  MoveL 10727 to (516.24, 531.44, 196) mm, rotated rx 180 ry 0 rz 160 deg; joints [9.799, 52.22, -5.839, -141.654, 53.227, 154.66]
  Set speed (17.9 mm/s)
  Call Extruder(1433.21511)
  MoveL 10728 to (515.75, 531.68, 196) mm, rotated rx -180 ry 0 rz 160 deg; joints [9.838, 52.138, -5.688, -141.642, 53.298, 154.686]
  Set speed (17.9 mm/s)
  Call Extruder(1436.45170)
  MoveL 10729 to (514.83, 532.12, 196) mm, rotated rx 180 ry 0 rz 160 deg; joints [9.91, 51.981, -5.403, -141.62, 53.429, 154.738]
  Set speed (17.9 mm/s)
  Call Extruder(1440.77463)
  MoveL 10730 to (513.57, 532.68, 196) mm, rotated rx -180 ry 0 rz 160 deg; joints [10.002, 51.769, -5.017, -141.596, 53.605, 154.81]
  Set speed (17.9 mm/s)
  Call Extruder(1445.24376)
  MoveL 10731 to (512.25, 533.19, 196) mm, rotated rx -180 ry 0 rz 160 deg; joints [10.092, 51.546, -4.609, -141.579, 53.788, 154.892]
  Set speed (17.9 mm/s)
  Call Extruder(1449.94818)
  MoveL 10732 to (510.84, 533.68, 196) mm, rotated rx 180 ry 0 rz 160 deg; joints [10.181, 51.306, -4.172, -141.568, 53.98, 154.985]
  Set speed (17.9 mm/s)
  Call Extruder(1452.28530)
  MoveL 10733 to (510.14, 533.89, 196) mm, rotated rx 180 ry 0 rz 160 deg; joints [10.223, 51.185, -3.952, -141.567, 54.075, 155.034]
  Set speed (17.9 mm/s)
  Call Extruder(1454.80660)
  MoveL 10734 to (509.37, 534.12, 196) mm, rotated rx 180 ry 0 rz 160 deg; joints [10.266, 51.054, -3.714, -141.566, 54.177, 155.088]
  Set speed (17.9 mm/s)
  Call Extruder(1459.03894)
  MoveL 10735 to (508.07, 534.45, 196) mm, rotated rx 180 ry 0 rz 160 deg; joints [10.335, 50.831, -3.309, -141.571, 54.349, 155.182]
  Set speed (17.9 mm/s)
  Call Extruder(1463.69218)
  MoveL 10736 to (506.63, 534.75, 196) mm, rotated rx -180 ry 0 rz 160 deg; joints [10.404, 50.584, -2.858, -141.584, 54.537, 155.292]
  Call Extruder(1468.33973)
  MoveL 10737 to (505.18, 535, 196) mm, rotated rx -180 ry 0 rz 160 deg; joints [10.467, 50.333, -2.403, -141.605, 54.724, 155.408]
  Call Extruder(1472.73701)
  MoveL 10738 to (503.8, 535.18, 196) mm, rotated rx -180 ry 0 rz 160 deg; joints [10.52, 50.094, -1.969, -141.631, 54.898, 155.523]
  Set speed (17.9 mm/s)
  Call Extruder(1477.45397)
  MoveL 10739 to (502.31, 535.3, 196) mm, rotated rx 180 ry 0 rz 160 deg; joints [10.569, 49.836, -1.5, -141.668, 55.084, 155.651]
  Set speed (17.9 mm/s)
  Call Extruder(1482.07202)
  MoveL 10740 to (500.85, 535.37, 196) mm, rotated rx 180 ry 0 rz 160 deg; joints [10.611, 49.582, -1.039, -141.711, 55.264, 155.781]
  Set speed (17.9 mm/s)
  Call Extruder(1486.54739)
  MoveL 10741 to (499.43, 535.38, 196) mm, rotated rx 180 ry 0 rz 160 deg; joints [10.644, 49.334, -0.59, -141.76, 55.436, 155.911]
  Set speed (10.0 mm/s)
  MoveL 10742 to (499.43, 535.38, 200) mm, rotated rx -180 ry 0 rz 160 deg; joints [10.644, 48.828, -0.582, -141.545, 55.045, 155.535]
  Set speed (120.0 mm/s)
  MoveL 10743 to (500.03, 535.97, 200) mm, rotated rx 180 ry 0 rz 160 deg; joints [10.704, 48.952, -0.806, -141.436, 54.992, 155.421]
  Set speed (19.5 mm/s)
  Call Extruder(1491.54324)
  MoveL 10744 to (498.3, 535.93, 200) mm, rotated rx 180 ry 0 rz 160 deg; joints [10.739, 48.648, -0.258, -141.503, 55.197, 155.584]
  Set speed (19.5 mm/s)
  Call Extruder(1494.78231)
  MoveL 10745 to (497.19, 535.86, 200) mm, rotated rx 180 ry 0 rz 160 deg; joints [10.756, 48.451, 0.097, -141.552, 55.328, 155.693]
  Set speed (19.5 mm/s)
  Call Extruder(1496.49093)
  MoveL 10746 to (496.6, 535.81, 200) mm, rotated rx -180 ry 0 rz 160 deg; joints [10.764, 48.347, 0.284, -141.579, 55.396, 155.751]
  Call Extruder(1498.85251)
  MoveL 10747 to (495.79, 535.72, 200) mm, rotated rx -180 ry 0 rz 160 deg; joints [10.772, 48.203, 0.543, -141.619, 55.489, 155.832]
  Set speed (19.5 mm/s)
  Call Extruder(1502.36924)
  MoveL 10748 to (494.59, 535.56, 200) mm, rotated rx -180 ry 0 rz 160 deg; joints [10.781, 47.99, 0.927, -141.682, 55.627, 155.955]
  Set speed (19.5 mm/s)
  Call Extruder(1507.13102)
  MoveL 10749 to (492.97, 535.28, 200) mm, rotated rx 180 ry 0 rz 160 deg; joints [10.784, 47.702, 1.445, -141.776, 55.809, 156.126]
  Set speed (19.5 mm/s)
  Call Extruder(1511.94509)
  MoveL 10750 to (491.35, 534.91, 200) mm, rotated rx -180 ry 0 rz 160 deg; joints [10.777, 47.412, 1.966, -141.88, 55.987, 156.302]
  Set speed (19.5 mm/s)
  Call Extruder(1515.30668)
  MoveL 10751 to (490.22, 534.61, 200) mm, rotated rx 180 ry 0 rz 160 deg; joints [10.766, 47.21, 2.328, -141.958, 56.109, 156.428]
  Set speed (19.5 mm/s)
  Call Extruder(1516.82836)
  MoveL 10752 to (489.72, 534.47, 200) mm, rotated rx 180 ry 0 rz 160 deg; joints [10.76, 47.12, 2.491, -141.995, 56.164, 156.485]
  Call Extruder(1519.31802)
  MoveL 10753 to (488.9, 534.21, 200) mm, rotated rx -180 ry 0 rz 160 deg; joints [10.747, 46.972, 2.756, -142.058, 56.251, 156.58]
  Set speed (19.5 mm/s)
  Call Extruder(1522.70288)
  MoveL 10754 to (487.79, 533.84, 200) mm, rotated rx -180 ry 0 rz 160 deg; joints [10.726, 46.772, 3.114, -142.145, 56.368, 156.71]
  Set speed (19.5 mm/s)
  Call Extruder(1527.20077)
  MoveL 10755 to (486.34, 533.28, 200) mm, rotated rx -180 ry 0 rz 160 deg; joints [10.69, 46.509, 3.586, -142.27, 56.518, 156.885]
  Set speed (19.5 mm/s)
  Call Extruder(1532.16103)
  MoveL 10756 to (484.77, 532.59, 200) mm, rotated rx 180 ry 0 rz 160 deg; joints [10.64, 46.223, 4.098, -142.417, 56.678, 157.081]
  Set speed (19.5 mm/s)
  Call Extruder(1535.74782)
  MoveL 10757 to (483.66, 532.04, 200) mm, rotated rx -180 ry 0 rz 160 deg; joints [10.597, 46.019, 4.463, -142.528, 56.789, 157.225]
  Set speed (19.5 mm/s)
  Call Extruder(1537.52530)
  MoveL 10758 to (483.11, 531.76, 200) mm, rotated rx 180 ry 0 rz 160 deg; joints [10.574, 45.919, 4.642, -142.585, 56.843, 157.296]
  Set speed (19.5 mm/s)
  Call Extruder(1539.75504)
  MoveL 10759 to (482.44, 531.39, 200) mm, rotated rx -180 ry 0 rz 160 deg; joints [10.542, 45.794, 4.865, -142.659, 56.908, 157.386]
  Set speed (19.5 mm/s)
  Call Extruder(1543.11777)
  MoveL 10760 to (481.43, 530.81, 200) mm, rotated rx -180 ry 0 rz 160 deg; joints [10.492, 45.608, 5.197, -142.772, 57.006, 157.522]
  Set speed (19.5 mm/s)
  Call Extruder(1547.76811)
  MoveL 10761 to (480.07, 529.95, 200) mm, rotated rx -180 ry 0 rz 160 deg; joints [10.413, 45.356, 5.647, -142.936, 57.134, 157.712]
  Call Extruder(1552.96193)
  MoveL 10762 to (478.61, 528.92, 200) mm, rotated rx 180 ry 0 rz 160 deg; joints [10.315, 45.082, 6.138, -143.128, 57.269, 157.925]
  Set speed (19.5 mm/s)
  Call Extruder(1556.13855)
  MoveL 10763 to (477.74, 528.25, 200) mm, rotated rx -180 ry 0 rz 160 deg; joints [10.248, 44.918, 6.429, -143.251, 57.346, 158.056]
  Set speed (19.5 mm/s)
  Call Extruder(1557.91549)
  MoveL 10764 to (477.26, 527.86, 200) mm, rotated rx 180 ry 0 rz 160 deg; joints [10.21, 44.828, 6.591, -143.321, 57.389, 158.129]
  Set speed (19.5 mm/s)
  Call Extruder(1560.20062)
  MoveL 10765 to (476.65, 527.36, 200) mm, rotated rx 180 ry 0 rz 160 deg; joints [10.158, 44.713, 6.795, -143.412, 57.442, 158.223]
  Set speed (19.5 mm/s)
  Call Extruder(1562.87061)
  MoveL 10766 to (475.96, 526.75, 200) mm, rotated rx 180 ry 0 rz 160 deg; joints [10.095, 44.581, 7.031, -143.521, 57.501, 158.334]
  Set speed (19.5 mm/s)
  Call Extruder(1564.37884)
  MoveL 10767 to (475.57, 526.4, 200) mm, rotated rx 180 ry 0 rz 160 deg; joints [10.058, 44.507, 7.162, -143.583, 57.534, 158.396]
  Set speed (19.5 mm/s)
  Call Extruder(1568.43038)
  MoveL 10768 to (474.56, 525.43, 200) mm, rotated rx -180 ry 0 rz 160 deg; joints [9.955, 44.314, 7.506, -143.753, 57.618, 158.563]
  Call Extruder(0.00000)
  Call Extruder(4.02287)
  MoveL 10769 to (473.6, 524.43, 200) mm, rotated rx 180 ry 0 rz 160 deg; joints [9.845, 44.128, 7.837, -143.929, 57.695, 158.729]
  Set speed (19.5 mm/s)
  Call Extruder(8.21913)
  MoveL 10770 to (472.64, 523.35, 200) mm, rotated rx 180 ry 0 rz 160 deg; joints [9.724, 43.941, 8.169, -144.116, 57.769, 158.901]
  Set speed (19.5 mm/s)
  Call Extruder(10.05952)
  MoveL 10771 to (472.23, 522.86, 200) mm, rotated rx 180 ry 0 rz 160 deg; joints [9.669, 43.861, 8.312, -144.2, 57.8, 158.977]
  Set speed (19.5 mm/s)
  Call Extruder(12.26771)
  MoveL 10772 to (471.75, 522.27, 200) mm, rotated rx 180 ry 0 rz 160 deg; joints [9.601, 43.767, 8.48, -144.301, 57.835, 159.067]
  Set speed (19.5 mm/s)
  Call Extruder(15.74515)
  MoveL 10773 to (471.02, 521.32, 200) mm, rotated rx 180 ry 0 rz 160 deg; joints [9.492, 43.622, 8.737, -144.464, 57.887, 159.209]
  Set speed (19.5 mm/s)
  Call Extruder(20.45172)
  MoveL 10774 to (470.09, 519.98, 200) mm, rotated rx 180 ry 0 rz 160 deg; joints [9.335, 43.435, 9.069, -144.689, 57.951, 159.4]
  Set speed (19.5 mm/s)
  Call Extruder(25.46049)
  MoveL 10775 to (469.17, 518.52, 200) mm, rotated rx 180 ry 0 rz 160 deg; joints [9.16, 43.246, 9.403, -144.935, 58.008, 159.602]
  Set speed (19.5 mm/s)
  Call Extruder(28.63180)
  MoveL 10776 to (468.62, 517.57, 200) mm, rotated rx 180 ry 0 rz 160 deg; joints [9.045, 43.133, 9.604, -145.093, 58.04, 159.728]
  Set speed (19.5 mm/s)
  Call Extruder(30.52229)
  MoveL 10777 to (468.3, 517, 200) mm, rotated rx -180 ry 0 rz 160 deg; joints [8.976, 43.068, 9.721, -145.188, 58.058, 159.803]
  Set speed (19.5 mm/s)
  Call Extruder(32.70849)
  MoveL 10778 to (467.95, 516.33, 200) mm, rotated rx -180 ry 0 rz 160 deg; joints [8.893, 42.995, 9.85, -145.3, 58.076, 159.889]
  Call Extruder(36.10735)
  MoveL 10779 to (467.43, 515.28, 200) mm, rotated rx 180 ry 0 rz 160 deg; joints [8.763, 42.884, 10.046, -145.474, 58.101, 160.022]
  Set speed (19.5 mm/s)
  Call Extruder(40.92807)
  MoveL 10780 to (466.76, 513.75, 200) mm, rotated rx -180 ry 0 rz 160 deg; joints [8.572, 42.739, 10.304, -145.725, 58.129, 160.209]
  Set speed (19.5 mm/s)
  Call Extruder(45.01848)
  MoveL 10781 to (466.25, 512.44, 200) mm, rotated rx -180 ry 0 rz 160 deg; joints [8.405, 42.625, 10.505, -145.941, 58.145, 160.365]
  Set speed (19.5 mm/s)
  Call Extruder(49.10868)
  MoveL 10782 to (465.79, 511.11, 200) mm, rotated rx -180 ry 0 rz 160 deg; joints [8.234, 42.52, 10.691, -146.159, 58.155, 160.518]
  Set speed (19.5 mm/s)
  Call Extruder(51.23461)
  MoveL 10783 to (465.57, 510.4, 200) mm, rotated rx -180 ry 0 rz 160 deg; joints [8.143, 42.468, 10.783, -146.273, 58.158, 160.597]
  Set speed (19.5 mm/s)
  Call Extruder(53.12982)
  MoveL 10784 to (465.39, 509.78, 200) mm, rotated rx -180 ry 0 rz 160 deg; joints [8.062, 42.425, 10.86, -146.375, 58.159, 160.667]
  Set speed (19.5 mm/s)
  Call Extruder(56.73452)
  MoveL 10785 to (465.06, 508.57, 200) mm, rotated rx 180 ry 0 rz 160 deg; joints [7.905, 42.345, 11, -146.57, 58.158, 160.799]
  Set speed (19.5 mm/s)
  Call Extruder(61.51678)
  MoveL 10786 to (464.71, 506.96, 200) mm, rotated rx 180 ry 0 rz 160 deg; joints [7.692, 42.253, 11.164, -146.831, 58.148, 160.969]
  Set speed (19.5 mm/s)
  Call Extruder(65.39166)
  MoveL 10787 to (464.48, 505.64, 200) mm, rotated rx -180 ry 0 rz 160 deg; joints [7.517, 42.188, 11.279, -147.043, 58.133, 161.104]
  Set speed (19.5 mm/s)
  Call Extruder(69.58261)
  MoveL 10788 to (464.28, 504.21, 200) mm, rotated rx -180 ry 0 rz 160 deg; joints [7.326, 42.126, 11.387, -147.272, 58.111, 161.247]
  Set speed (19.5 mm/s)
  Call Extruder(71.46441)
  MoveL 10789 to (464.21, 503.56, 200) mm, rotated rx -180 ry 0 rz 160 deg; joints [7.239, 42.102, 11.431, -147.376, 58.099, 161.31]
  Set speed (19.5 mm/s)
  Call Extruder(73.67117)
  MoveL 10790 to (464.14, 502.81, 200) mm, rotated rx -180 ry 0 rz 160 deg; joints [7.136, 42.076, 11.477, -147.497, 58.083, 161.384]
  Set speed (19.5 mm/s)
  Call Extruder(77.06464)
  MoveL 10791 to (464.06, 501.64, 200) mm, rotated rx 180 ry 0 rz 160 deg; joints [6.979, 42.04, 11.54, -147.682, 58.056, 161.494]
  Set speed (19.5 mm/s)
  Call Extruder(81.77489)
  MoveL 10792 to (464.03, 500.01, 200) mm, rotated rx -180 ry 0 rz 160 deg; joints [6.757, 42.003, 11.605, -147.939, 58.01, 161.643]
  Set speed (19.5 mm/s)
  Call Extruder(86.94228)
  MoveL 10793 to (464.07, 498.23, 200) mm, rotated rx 180 ry 0 rz 160 deg; joints [6.512, 41.977, 11.652, -148.22, 57.95, 161.801]
  Set speed (19.5 mm/s)
  Call Extruder(89.93783)
  MoveL 10794 to (464.14, 497.19, 200) mm, rotated rx -180 ry 0 rz 160 deg; joints [6.37, 41.969, 11.665, -148.382, 57.911, 161.89]
  Set speed (19.5 mm/s)
  Call Extruder(91.84959)
  MoveL 10795 to (464.2, 496.54, 200) mm, rotated rx -180 ry 0 rz 160 deg; joints [6.279, 41.966, 11.67, -148.485, 57.884, 161.945]
  Set speed (19.5 mm/s)
  Call Extruder(94.05179)
  MoveL 10796 to (464.28, 495.78, 200) mm, rotated rx 180 ry 0 rz 160 deg; joints [6.174, 41.966, 11.67, -148.602, 57.852, 162.008]
  Set speed (19.5 mm/s)
  Call Extruder(97.68286)
  MoveL 10797 to (464.44, 494.54, 200) mm, rotated rx 180 ry 0 rz 160 deg; joints [6.001, 41.971, 11.661, -148.795, 57.796, 162.109]
  Set speed (19.5 mm/s)
  Call Extruder(102.26103)
  MoveL 10798 to (464.72, 492.98, 200) mm, rotated rx 180 ry 0 rz 160 deg; joints [5.784, 41.989, 11.63, -149.035, 57.717, 162.23]
  Set speed (19.5 mm/s)
  Call Extruder(107.32984)
  MoveL 10799 to (465.1, 491.27, 200) mm, rotated rx -180 ry 0 rz 160 deg; joints [5.545, 42.024, 11.568, -149.296, 57.621, 162.358]
  Set speed (19.5 mm/s)
  Call Extruder(110.39224)
  MoveL 10800 to (465.38, 490.25, 200) mm, rotated rx 180 ry 0 rz 160 deg; joints [5.402, 42.053, 11.518, -149.451, 57.559, 162.432]
  Set speed (19.5 mm/s)
  Call Extruder(112.51019)
  MoveL 10801 to (465.58, 489.55, 200) mm, rotated rx 180 ry 0 rz 160 deg; joints [5.303, 42.075, 11.479, -149.557, 57.515, 162.482]
  Set speed (19.5 mm/s)
  Call Extruder(114.48994)
  MoveL 10802 to (465.79, 488.9, 200) mm, rotated rx 180 ry 0 rz 160 deg; joints [5.211, 42.098, 11.437, -149.655, 57.472, 162.527]
  Set speed (19.5 mm/s)
  Call Extruder(118.61417)
  MoveL 10803 to (466.25, 487.56, 200) mm, rotated rx -180 ry 0 rz 160 deg; joints [5.022, 42.154, 11.338, -149.856, 57.378, 162.617]
  Set speed (19.5 mm/s)
  Call Extruder(122.74688)
  MoveL 10804 to (466.77, 486.23, 200) mm, rotated rx 180 ry 0 rz 160 deg; joints [4.834, 42.219, 11.224, -150.053, 57.279, 162.702]
  Set speed (19.5 mm/s)
  Call Extruder(127.54821)
  MoveL 10805 to (467.44, 484.71, 200) mm, rotated rx 180 ry 0 rz 160 deg; joints [4.619, 42.306, 11.069, -150.275, 57.157, 162.795]
  Set speed (19.5 mm/s)
  Call Extruder(130.89563)
  MoveL 10806 to (467.96, 483.67, 200) mm, rotated rx 180 ry 0 rz 160 deg; joints [4.472, 42.376, 10.945, -150.425, 57.067, 162.854]
  Set speed (19.5 mm/s)
  Call Extruder(132.98107)
  MoveL 10807 to (468.29, 483.03, 200) mm, rotated rx 180 ry 0 rz 160 deg; joints [4.381, 42.422, 10.865, -150.518, 57.009, 162.889]
  Set speed (19.5 mm/s)
  Call Extruder(134.98230)
  MoveL 10808 to (468.62, 482.43, 200) mm, rotated rx 180 ry 0 rz 160 deg; joints [4.295, 42.468, 10.783, -150.604, 56.953, 162.922]
  Call Extruder(138.15507)
  MoveL 10809 to (469.17, 481.48, 200) mm, rotated rx 180 ry 0 rz 160 deg; joints [4.16, 42.546, 10.646, -150.739, 56.862, 162.971]
  Set speed (19.5 mm/s)
  Call Extruder(143.17117)
  MoveL 10810 to (470.09, 480.01, 200) mm, rotated rx 180 ry 0 rz 160 deg; joints [3.951, 42.678, 10.41, -150.945, 56.711, 163.042]
  Set speed (19.5 mm/s)
  Call Extruder(148.38694)
  MoveL 10811 to (471.14, 478.54, 200) mm, rotated rx 180 ry 0 rz 160 deg; joints [3.742, 42.832, 10.139, -151.147, 56.547, 163.105]
  Set speed (19.5 mm/s)
  Call Extruder(151.29556)
  MoveL 10812 to (471.75, 477.74, 200) mm, rotated rx -180 ry 0 rz 160 deg; joints [3.629, 42.923, 9.977, -151.255, 56.452, 163.136]
  Call Extruder(153.54810)
  MoveL 10813 to (472.23, 477.14, 200) mm, rotated rx 180 ry 0 rz 160 deg; joints [3.542, 42.996, 9.848, -151.336, 56.377, 163.159]
  Call Extruder(155.46198)
  MoveL 10814 to (472.66, 476.63, 200) mm, rotated rx 180 ry 0 rz 160 deg; joints [3.471, 43.06, 9.733, -151.403, 56.313, 163.176]
  Set speed (19.5 mm/s)
  Call Extruder(158.59926)
  MoveL 10815 to (473.37, 475.82, 200) mm, rotated rx -180 ry 0 rz 160 deg; joints [3.355, 43.169, 9.541, -151.509, 56.206, 163.202]
  Set speed (19.5 mm/s)
  Call Extruder(163.56171)
  MoveL 10816 to (474.56, 474.58, 200) mm, rotated rx -180 ry 0 rz 160 deg; joints [3.178, 43.351, 9.218, -151.668, 56.031, 163.235]
  Call Extruder(168.35793)
  MoveL 10817 to (475.75, 473.43, 200) mm, rotated rx 180 ry 0 rz 160 deg; joints [3.015, 43.537, 8.888, -151.81, 55.857, 163.258]
  Set speed (19.5 mm/s)
  Call Extruder(171.81964)
  MoveL 10818 to (476.65, 472.64, 200) mm, rotated rx -180 ry 0 rz 160 deg; joints [2.903, 43.678, 8.637, -151.904, 55.728, 163.268]
  Set speed (19.5 mm/s)
  Call Extruder(173.98588)
  MoveL 10819 to (477.23, 472.16, 200) mm, rotated rx 180 ry 0 rz 160 deg; joints [2.835, 43.769, 8.476, -151.961, 55.646, 163.272]
  Set speed (19.5 mm/s)
  Call Extruder(175.90921)
  MoveL 10820 to (477.74, 471.75, 200) mm, rotated rx -180 ry 0 rz 160 deg; joints [2.776, 43.851, 8.33, -152.009, 55.573, 163.275]
  Call Extruder(179.09732)
  MoveL 10821 to (478.62, 471.08, 200) mm, rotated rx 180 ry 0 rz 160 deg; joints [2.68, 43.99, 8.083, -152.085, 55.45, 163.276]
  Set speed (19.5 mm/s)
  Call Extruder(183.97603)
  MoveL 10822 to (480, 470.11, 200) mm, rotated rx -180 ry 0 rz 160 deg; joints [2.543, 44.211, 7.69, -152.19, 55.258, 163.27]
  Set speed (19.5 mm/s)
  Call Extruder(189.20423)
  MoveL 10823 to (481.52, 469.14, 200) mm, rotated rx -180 ry 0 rz 160 deg; joints [2.405, 44.457, 7.251, -152.287, 55.048, 163.252]
  Set speed (19.5 mm/s)
  Call Extruder(192.27016)
  MoveL 10824 to (482.44, 468.61, 200) mm, rotated rx 180 ry 0 rz 160 deg; joints [2.33, 44.606, 6.985, -152.337, 54.923, 163.236]
  Set speed (19.5 mm/s)
  Call Extruder(194.46720)
  MoveL 10825 to (483.1, 468.25, 200) mm, rotated rx -180 ry 0 rz 160 deg; joints [2.279, 44.715, 6.792, -152.37, 54.833, 163.223]
  Set speed (19.5 mm/s)
  Call Extruder(196.26423)
  MoveL 10826 to (483.65, 467.96, 200) mm, rotated rx 180 ry 0 rz 160 deg; joints [2.238, 44.805, 6.631, -152.395, 54.759, 163.21]
  Set speed (19.5 mm/s)
  Call Extruder(199.39284)
  MoveL 10827 to (484.62, 467.49, 200) mm, rotated rx -180 ry 0 rz 160 deg; joints [2.17, 44.964, 6.347, -152.433, 54.628, 163.185]
  Set speed (19.5 mm/s)
  Call Extruder(204.45409)
  MoveL 10828 to (486.22, 466.77, 200) mm, rotated rx -180 ry 0 rz 160 deg; joints [2.069, 45.228, 5.876, -152.484, 54.415, 163.137]
  Set speed (19.5 mm/s)
  Call Extruder(209.24454)
  MoveL 10829 to (487.76, 466.17, 200) mm, rotated rx -180 ry 0 rz 160 deg; joints [1.983, 45.485, 5.418, -152.519, 54.212, 163.081]
  Set speed (19.5 mm/s)
  Call Extruder(212.71224)
  MoveL 10830 to (488.9, 465.79, 200) mm, rotated rx 180 ry 0 rz 160 deg; joints [1.928, 45.674, 5.079, -152.534, 54.063, 163.034]
  Set speed (19.5 mm/s)
  Call Extruder(214.66020)
  MoveL 10831 to (489.54, 465.59, 200) mm, rotated rx 180 ry 0 rz 160 deg; joints [1.899, 45.782, 4.886, -152.54, 53.98, 163.006]
  Set speed (19.5 mm/s)
  Call Extruder(216.76262)
  MoveL 10832 to (490.24, 465.39, 200) mm, rotated rx -180 ry 0 rz 160 deg; joints [1.869, 45.899, 4.677, -152.544, 53.889, 162.974]
  Set speed (19.5 mm/s)
  Call Extruder(220.34143)
  MoveL 10833 to (491.43, 465.06, 200) mm, rotated rx -180 ry 0 rz 160 deg; joints [1.822, 46.101, 4.316, -152.546, 53.734, 162.916]
  Set speed (19.5 mm/s)
  Call Extruder(224.94326)
  MoveL 10834 to (492.98, 464.72, 200) mm, rotated rx 180 ry 0 rz 160 deg; joints [1.771, 46.364, 3.845, -152.535, 53.534, 162.833]
  Set speed (19.5 mm/s)
  Call Extruder(229.90057)
  MoveL 10835 to (494.67, 464.43, 200) mm, rotated rx -180 ry 0 rz 160 deg; joints [1.727, 46.653, 3.328, -152.51, 53.319, 162.733]
  Set speed (19.5 mm/s)
  Call Extruder(233.17180)
  MoveL 10836 to (495.79, 464.28, 200) mm, rotated rx 180 ry 0 rz 160 deg; joints [1.704, 46.845, 2.983, -152.485, 53.177, 162.662]
  Call Extruder(235.17639)
  MoveL 10837 to (496.48, 464.2, 200) mm, rotated rx -180 ry 0 rz 160 deg; joints [1.691, 46.963, 2.771, -152.468, 53.09, 162.616]
  Call Extruder(237.23430)
  MoveL 10838 to (497.19, 464.14, 200) mm, rotated rx 180 ry 0 rz 160 deg; joints [1.681, 47.085, 2.552, -152.447, 53, 162.568]
  Set speed (19.5 mm/s)
  Call Extruder(241.26374)
  MoveL 10839 to (498.57, 464.06, 200) mm, rotated rx 180 ry 0 rz 160 deg; joints [1.665, 47.326, 2.12, -152.399, 52.826, 162.468]
  Set speed (19.5 mm/s)
  Call Extruder(245.57319)
  MoveL 10840 to (500.06, 464.03, 200) mm, rotated rx -180 ry 0 rz 160 deg; joints [1.655, 47.585, 1.655, -152.337, 52.641, 162.355]
  Set speed (19.5 mm/s)
  Call Extruder(250.17367)
  MoveL 10841 to (501.65, 464.07, 200) mm, rotated rx 180 ry 0 rz 160 deg; joints [1.654, 47.863, 1.155, -152.259, 52.444, 162.226]
  Set speed (19.5 mm/s)
  Call Extruder(253.55314)
  MoveL 10842 to (502.81, 464.14, 200) mm, rotated rx 180 ry 0 rz 160 deg; joints [1.66, 48.068, 0.787, -152.194, 52.301, 162.126]
  Set speed (19.5 mm/s)
  Call Extruder(255.72148)
  MoveL 10843 to (503.56, 464.21, 200) mm, rotated rx -180 ry 0 rz 160 deg; joints [1.665, 48.2, 0.549, -152.149, 52.209, 162.059]
  Set speed (19.5 mm/s)
  Call Extruder(257.62118)
  MoveL 10844 to (504.21, 464.28, 200) mm, rotated rx -180 ry 0 rz 160 deg; joints [1.672, 48.316, 0.341, -152.107, 52.13, 161.999]
  Set speed (19.5 mm/s)
  Call Extruder(261.27000)
  MoveL 10845 to (505.46, 464.44, 200) mm, rotated rx -180 ry 0 rz 160 deg; joints [1.688, 48.538, -0.059, -152.023, 51.978, 161.882]
  Call Extruder(265.80352)
  MoveL 10846 to (507, 464.72, 200) mm, rotated rx 180 ry 0 rz 160 deg; joints [1.717, 48.813, -0.555, -151.907, 51.791, 161.729]
  Set speed (19.5 mm/s)
  Call Extruder(270.83135)
  MoveL 10847 to (508.7, 465.1, 200) mm, rotated rx 180 ry 0 rz 160 deg; joints [1.758, 49.118, -1.106, -151.766, 51.588, 161.55]
  Set speed (19.5 mm/s)
  Call Extruder(274.04053)
  MoveL 10848 to (509.77, 465.39, 200) mm, rotated rx 180 ry 0 rz 160 deg; joints [1.79, 49.312, -1.456, -151.669, 51.461, 161.432]
  Call Extruder(275.88445)
  MoveL 10849 to (510.38, 465.56, 200) mm, rotated rx 180 ry 0 rz 160 deg; joints [1.809, 49.424, -1.656, -151.611, 51.389, 161.363]
  Set speed (19.5 mm/s)
  Call Extruder(278.06632)
  MoveL 10850 to (511.1, 465.79, 200) mm, rotated rx -180 ry 0 rz 160 deg; joints [1.835, 49.555, -1.893, -151.54, 51.304, 161.279]
  Call Extruder(281.26040)
  MoveL 10851 to (512.15, 466.14, 200) mm, rotated rx 180 ry 0 rz 160 deg; joints [1.874, 49.746, -2.238, -151.433, 51.181, 161.155]
  Set speed (19.5 mm/s)
  Call Extruder(286.32736)
  MoveL 10852 to (513.78, 466.77, 200) mm, rotated rx -180 ry 0 rz 160 deg; joints [1.946, 50.047, -2.782, -151.252, 50.991, 160.951]
  Set speed (19.5 mm/s)
  Call Extruder(290.33252)
  MoveL 10853 to (515.05, 467.33, 200) mm, rotated rx 180 ry 0 rz 160 deg; joints [2.009, 50.282, -3.206, -151.101, 50.846, 160.784]
  Set speed (19.5 mm/s)
  Call Extruder(294.49619)
  MoveL 10854 to (516.34, 467.96, 200) mm, rotated rx 180 ry 0 rz 160 deg; joints [2.081, 50.523, -3.642, -150.936, 50.699, 160.607]
  Set speed (19.5 mm/s)
  Call Extruder(296.55530)
  MoveL 10855 to (516.97, 468.29, 200) mm, rotated rx -180 ry 0 rz 160 deg; joints [2.118, 50.641, -3.857, -150.853, 50.628, 160.518]
  Call Extruder(298.51486)
  MoveL 10856 to (517.56, 468.61, 200) mm, rotated rx -180 ry 0 rz 160 deg; joints [2.155, 50.753, -4.059, -150.771, 50.561, 160.432]
  Set speed (19.5 mm/s)
  Call Extruder(302.61005)
  MoveL 10857 to (518.78, 469.33, 200) mm, rotated rx -180 ry 0 rz 160 deg; joints [2.237, 50.984, -4.477, -150.596, 50.426, 160.25]
  Set speed (19.5 mm/s)
  Call Extruder(306.74297)
  MoveL 10858 to (519.99, 470.09, 200) mm, rotated rx -180 ry 0 rz 160 deg; joints [2.325, 51.213, -4.893, -150.413, 50.293, 160.063]
  Set speed (19.5 mm/s)
  Call Extruder(311.71130)
  MoveL 10859 to (521.39, 471.08, 200) mm, rotated rx -180 ry 0 rz 160 deg; joints [2.438, 51.483, -5.382, -150.184, 50.142, 159.832]
  Set speed (19.5 mm/s)
  Call Extruder(314.86599)
  MoveL 10860 to (522.25, 471.75, 200) mm, rotated rx 180 ry 0 rz 160 deg; joints [2.514, 51.651, -5.686, -150.034, 50.05, 159.684]
  Call Extruder(316.95477)
  MoveL 10861 to (522.82, 472.2, 200) mm, rotated rx 180 ry 0 rz 160 deg; joints [2.566, 51.76, -5.885, -149.933, 49.991, 159.585]
  Set speed (19.5 mm/s)
  Call Extruder(318.95555)
  MoveL 10862 to (523.35, 472.64, 200) mm, rotated rx 180 ry 0 rz 160 deg; joints [2.617, 51.864, -6.072, -149.835, 49.935, 159.49]
  Set speed (19.5 mm/s)
  Call Extruder(323.14808)
  MoveL 10863 to (524.43, 473.6, 200) mm, rotated rx -180 ry 0 rz 160 deg; joints [2.726, 52.077, -6.46, -149.627, 49.824, 159.289]
  Set speed (19.5 mm/s)
  Call Extruder(327.13768)
  MoveL 10864 to (525.43, 474.55, 200) mm, rotated rx 180 ry 0 rz 160 deg; joints [2.835, 52.275, -6.819, -149.425, 49.723, 159.096]
  Set speed (19.5 mm/s)
  Call Extruder(332.13186)
  MoveL 10865 to (526.62, 475.81, 200) mm, rotated rx -180 ry 0 rz 160 deg; joints [2.979, 52.514, -7.253, -149.165, 49.607, 158.851]
  Set speed (19.5 mm/s)
  Call Extruder(335.34961)
  MoveL 10866 to (527.35, 476.64, 200) mm, rotated rx -180 ry 0 rz 160 deg; joints [3.074, 52.663, -7.524, -148.994, 49.537, 158.693]
  Set speed (19.5 mm/s)
  Call Extruder(337.34953)
  MoveL 10867 to (527.79, 477.17, 200) mm, rotated rx 180 ry 0 rz 160 deg; joints [3.135, 52.754, -7.689, -148.887, 49.496, 158.595]
  Set speed (19.5 mm/s)
  Call Extruder(339.44281)
  MoveL 10868 to (528.25, 477.74, 200) mm, rotated rx -180 ry 0 rz 160 deg; joints [3.199, 52.847, -7.858, -148.775, 49.454, 158.492]
  Set speed (19.5 mm/s)
  Call Extruder(343.49847)
  MoveL 10869 to (529.09, 478.85, 200) mm, rotated rx 180 ry 0 rz 160 deg; joints [3.327, 53.022, -8.177, -148.555, 49.379, 158.292]
  Set speed (19.5 mm/s)
  Call Extruder(347.67724)
  MoveL 10870 to (529.92, 480.03, 200) mm, rotated rx 180 ry 0 rz 160 deg; joints [3.462, 53.196, -8.493, -148.325, 49.308, 158.086]
  Set speed (19.5 mm/s)
  Call Extruder(352.76875)
  MoveL 10871 to (530.86, 481.52, 200) mm, rotated rx 180 ry 0 rz 160 deg; joints [3.632, 53.396, -8.857, -148.043, 49.232, 157.836]
  Set speed (19.5 mm/s)
  Call Extruder(355.84628)
  MoveL 10872 to (531.39, 482.44, 200) mm, rotated rx 180 ry 0 rz 160 deg; joints [3.737, 53.511, -9.066, -147.871, 49.192, 157.686]
  Call Extruder(357.82949)
  MoveL 10873 to (531.72, 483.04, 200) mm, rotated rx 180 ry 0 rz 160 deg; joints [3.806, 53.583, -9.198, -147.76, 49.168, 157.589]
  Set speed (19.5 mm/s)
  Call Extruder(359.84338)
  MoveL 10874 to (532.04, 483.66, 200) mm, rotated rx 180 ry 0 rz 160 deg; joints [3.877, 53.654, -9.327, -147.646, 49.146, 157.492]
  Set speed (19.5 mm/s)
  Call Extruder(363.38135)
  MoveL 10875 to (532.58, 484.75, 200) mm, rotated rx -180 ry 0 rz 160 deg; joints [4.002, 53.775, -9.547, -147.448, 49.11, 157.321]
  Set speed (19.5 mm/s)
  Call Extruder(368.11581)
  MoveL 10876 to (533.24, 486.25, 200) mm, rotated rx 180 ry 0 rz 160 deg; joints [4.173, 53.926, -9.821, -147.181, 49.072, 157.096]
  Call Extruder(372.16412)
  MoveL 10877 to (533.75, 487.55, 200) mm, rotated rx 180 ry 0 rz 160 deg; joints [4.322, 54.044, -10.037, -146.953, 49.049, 156.907]
  Set speed (19.5 mm/s)
  Call Extruder(376.25069)
  MoveL 10878 to (534.2, 488.88, 200) mm, rotated rx -180 ry 0 rz 160 deg; joints [4.475, 54.155, -10.239, -146.724, 49.033, 156.719]
  Set speed (19.5 mm/s)
  Call Extruder(378.15464)
  MoveL 10879 to (534.4, 489.51, 200) mm, rotated rx 180 ry 0 rz 160 deg; joints [4.547, 54.204, -10.329, -146.617, 49.028, 156.632]
  Call Extruder(380.30431)
  MoveL 10880 to (534.61, 490.22, 200) mm, rotated rx -180 ry 0 rz 160 deg; joints [4.629, 54.257, -10.424, -146.496, 49.024, 156.535]
  Set speed (19.5 mm/s)
  Call Extruder(384.44251)
  MoveL 10881 to (534.97, 491.61, 200) mm, rotated rx -180 ry 0 rz 160 deg; joints [4.788, 54.351, -10.597, -146.266, 49.023, 156.352]
  Set speed (19.5 mm/s)
  Call Extruder(388.48294)
  MoveL 10882 to (535.28, 492.97, 200) mm, rotated rx -180 ry 0 rz 160 deg; joints [4.945, 54.434, -10.748, -146.043, 49.029, 156.176]
  Call Extruder(392.56836)
  MoveL 10883 to (535.52, 494.36, 200) mm, rotated rx -180 ry 0 rz 160 deg; joints [5.105, 54.508, -10.882, -145.819, 49.044, 156.004]
  Set speed (19.5 mm/s)
  Call Extruder(396.75907)
  MoveL 10884 to (535.72, 495.79, 200) mm, rotated rx 180 ry 0 rz 160 deg; joints [5.271, 54.573, -11, -145.593, 49.068, 155.833]
  Set speed (19.5 mm/s)
  Call Extruder(398.56129)
  MoveL 10885 to (535.79, 496.41, 200) mm, rotated rx 180 ry 0 rz 160 deg; joints [5.343, 54.598, -11.046, -145.496, 49.08, 155.761]
  Set speed (19.5 mm/s)
  Call Extruder(400.77767)
  MoveL 10886 to (535.86, 497.17, 200) mm, rotated rx 180 ry 0 rz 160 deg; joints [5.432, 54.626, -11.097, -145.378, 49.097, 155.674]
  Set speed (19.5 mm/s)
  Call Extruder(404.03086)
  MoveL 10887 to (535.93, 498.29, 200) mm, rotated rx -180 ry 0 rz 160 deg; joints [5.562, 54.662, -11.164, -145.206, 49.127, 155.548]
  Set speed (19.5 mm/s)
  Call Extruder(408.93794)
  MoveL 10888 to (535.97, 499.99, 200) mm, rotated rx 180 ry 0 rz 160 deg; joints [5.76, 54.704, -11.24, -144.951, 49.18, 155.366]
  Set speed (19.5 mm/s)
  Call Extruder(413.66743)
  MoveL 10889 to (535.94, 501.62, 200) mm, rotated rx -180 ry 0 rz 160 deg; joints [5.951, 54.731, -11.289, -144.711, 49.242, 155.2]
  Set speed (19.5 mm/s)
  Call Extruder(417.10827)
  MoveL 10890 to (535.86, 502.81, 200) mm, rotated rx 180 ry 0 rz 160 deg; joints [6.09, 54.74, -11.305, -144.54, 49.295, 155.085]
  Set speed (19.5 mm/s)
  Call Extruder(419.01492)
  MoveL 10891 to (535.8, 503.46, 200) mm, rotated rx -180 ry 0 rz 160 deg; joints [6.167, 54.742, -11.31, -144.447, 49.326, 155.023]
  Call Extruder(421.19666)
  MoveL 10892 to (535.72, 504.21, 200) mm, rotated rx 180 ry 0 rz 160 deg; joints [6.256, 54.742, -11.309, -144.341, 49.363, 154.955]
  Set speed (19.5 mm/s)
  Call Extruder(424.66076)
  MoveL 10893 to (535.56, 505.4, 200) mm, rotated rx 180 ry 0 rz 160 deg; joints [6.396, 54.737, -11.301, -144.175, 49.426, 154.849]
  Set speed (19.5 mm/s)
  Call Extruder(429.44750)
  MoveL 10894 to (535.28, 507.03, 200) mm, rotated rx -180 ry 0 rz 160 deg; joints [6.59, 54.718, -11.265, -143.953, 49.522, 154.711]
  Set speed (19.5 mm/s)
  Call Extruder(434.59312)
  MoveL 10895 to (534.88, 508.76, 200) mm, rotated rx 180 ry 0 rz 160 deg; joints [6.798, 54.68, -11.196, -143.722, 49.636, 154.575]
  Set speed (19.5 mm/s)
  Call Extruder(437.63190)
  MoveL 10896 to (534.61, 509.78, 200) mm, rotated rx 180 ry 0 rz 160 deg; joints [6.921, 54.65, -11.141, -143.589, 49.709, 154.501]
  Set speed (19.5 mm/s)
  Call Extruder(439.52391)
  MoveL 10897 to (534.43, 510.4, 200) mm, rotated rx -180 ry 0 rz 160 deg; joints [6.996, 54.629, -11.102, -143.508, 49.755, 154.456]
  Call Extruder(441.64529)
  MoveL 10898 to (534.21, 511.1, 200) mm, rotated rx -180 ry 0 rz 160 deg; joints [7.081, 54.602, -11.054, -143.419, 49.81, 154.409]
  Set speed (19.5 mm/s)
  Call Extruder(445.15058)
  MoveL 10899 to (533.82, 512.25, 200) mm, rotated rx 180 ry 0 rz 160 deg; joints [7.221, 54.554, -10.966, -143.275, 49.902, 154.334]
  Set speed (19.5 mm/s)
  Call Extruder(449.90569)
  MoveL 10900 to (533.23, 513.78, 200) mm, rotated rx 180 ry 0 rz 160 deg; joints [7.408, 54.475, -10.822, -143.087, 50.035, 154.243]
  Set speed (19.5 mm/s)
  Call Extruder(454.46983)
  MoveL 10901 to (532.6, 515.22, 200) mm, rotated rx 180 ry 0 rz 160 deg; joints [7.587, 54.387, -10.662, -142.914, 50.17, 154.165]
  Set speed (19.5 mm/s)
  Call Extruder(458.04411)
  MoveL 10902 to (532.05, 516.33, 200) mm, rotated rx -180 ry 0 rz 160 deg; joints [7.724, 54.308, -10.518, -142.785, 50.282, 154.113]
  Set speed (19.5 mm/s)
  Call Extruder(459.91073)
  MoveL 10903 to (531.75, 516.9, 200) mm, rotated rx 180 ry 0 rz 160 deg; joints [7.796, 54.265, -10.44, -142.719, 50.342, 154.088]
  Call Extruder(462.12577)
  MoveL 10904 to (531.38, 517.57, 200) mm, rotated rx -180 ry 0 rz 160 deg; joints [7.88, 54.211, -10.341, -142.643, 50.414, 154.06]
  Set speed (19.5 mm/s)
  Call Extruder(465.53486)
  MoveL 10905 to (530.79, 518.59, 200) mm, rotated rx 180 ry 0 rz 160 deg; joints [8.009, 54.124, -10.182, -142.529, 50.528, 154.021]
  Set speed (19.5 mm/s)
  Call Extruder(470.31085)
  MoveL 10906 to (529.91, 519.99, 200) mm, rotated rx 180 ry 0 rz 160 deg; joints [8.187, 53.989, -9.937, -142.377, 50.693, 153.977]
  Set speed (19.5 mm/s)
  Call Extruder(475.18781)
  MoveL 10907 to (528.94, 521.36, 200) mm, rotated rx 180 ry 0 rz 160 deg; joints [8.365, 53.839, -9.663, -142.233, 50.869, 153.944]
  Set speed (19.5 mm/s)
  Call Extruder(478.47209)
  MoveL 10908 to (528.25, 522.26, 200) mm, rotated rx -180 ry 0 rz 160 deg; joints [8.483, 53.73, -9.465, -142.141, 50.991, 153.928]
  Set speed (19.5 mm/s)
  Call Extruder(480.40498)
  MoveL 10909 to (527.83, 522.78, 200) mm, rotated rx -180 ry 0 rz 160 deg; joints [8.551, 53.664, -9.345, -142.089, 51.064, 153.921]
  Call Extruder(482.53860)
  MoveL 10910 to (527.36, 523.35, 200) mm, rotated rx 180 ry 0 rz 160 deg; joints [8.626, 53.589, -9.208, -142.033, 51.146, 153.916]
  Set speed (19.5 mm/s)
  Call Extruder(485.70352)
  MoveL 10911 to (526.64, 524.17, 200) mm, rotated rx 180 ry 0 rz 160 deg; joints [8.736, 53.474, -8.998, -141.953, 51.268, 153.911]
  Call Extruder(490.71750)
  MoveL 10912 to (525.45, 525.43, 200) mm, rotated rx -180 ry 0 rz 160 deg; joints [8.906, 53.282, -8.649, -141.836, 51.467, 153.914]
  Set speed (19.5 mm/s)
  Call Extruder(495.87147)
  MoveL 10913 to (524.15, 526.66, 200) mm, rotated rx -180 ry 0 rz 160 deg; joints [9.074, 53.072, -8.266, -141.727, 51.676, 153.93]
  Call Extruder(498.92301)
  MoveL 10914 to (523.36, 527.35, 200) mm, rotated rx 180 ry 0 rz 160 deg; joints [9.171, 52.941, -8.029, -141.668, 51.803, 153.945]
  Call Extruder(500.64178)
  MoveL 10915 to (522.9, 527.73, 200) mm, rotated rx -180 ry 0 rz 160 deg; joints [9.225, 52.866, -7.893, -141.636, 51.874, 153.955]
  Set speed (19.5 mm/s)
  Call Extruder(503.05292)
  MoveL 10916 to (522.26, 528.26, 200) mm, rotated rx 180 ry 0 rz 160 deg; joints [9.299, 52.759, -7.698, -141.594, 51.976, 153.972]
  Set speed (19.5 mm/s)
  Call Extruder(505.89885)
  MoveL 10917 to (521.48, 528.86, 200) mm, rotated rx 180 ry 0 rz 160 deg; joints [9.386, 52.63, -7.464, -141.547, 52.096, 153.995]
  Set speed (19.5 mm/s)
  Call Extruder(511.22646)
  MoveL 10918 to (519.97, 529.92, 200) mm, rotated rx 180 ry 0 rz 160 deg; joints [9.542, 52.38, -7.009, -141.468, 52.325, 154.047]
  Set speed (19.5 mm/s)
  Call Extruder(516.20964)
  MoveL 10919 to (518.52, 530.84, 200) mm, rotated rx -180 ry 0 rz 160 deg; joints [9.68, 52.135, -6.565, -141.407, 52.541, 154.108]
  Set speed (19.5 mm/s)
  Call Extruder(519.36088)
  MoveL 10920 to (517.57, 531.38, 200) mm, rotated rx -180 ry 0 rz 160 deg; joints [9.764, 51.977, -6.277, -141.373, 52.679, 154.152]
  Set speed (19.5 mm/s)
  Call Extruder(521.13560)
  MoveL 10921 to (517.04, 531.68, 200) mm, rotated rx 180 ry 0 rz 160 deg; joints [9.811, 51.886, -6.113, -141.356, 52.757, 154.178]
  Call Extruder(523.40110)
  MoveL 10922 to (516.34, 532.04, 200) mm, rotated rx 180 ry 0 rz 160 deg; joints [9.868, 51.769, -5.9, -141.336, 52.856, 154.214]
  Set speed (19.5 mm/s)
  Call Extruder(526.79979)
  MoveL 10923 to (515.29, 532.56, 200) mm, rotated rx -180 ry 0 rz 160 deg; joints [9.952, 51.591, -5.577, -141.31, 53.006, 154.27]
  Set speed (19.5 mm/s)
  Call Extruder(531.50603)
  MoveL 10924 to (513.8, 533.22, 200) mm, rotated rx 180 ry 0 rz 160 deg; joints [10.062, 51.338, -5.118, -141.282, 53.214, 154.356]
  Set speed (19.5 mm/s)
  Call Extruder(536.24163)
  MoveL 10925 to (512.28, 533.81, 200) mm, rotated rx 180 ry 0 rz 160 deg; joints [10.167, 51.077, -4.647, -141.263, 53.424, 154.451]
  Set speed (19.5 mm/s)
  Call Extruder(541.46898)
  MoveL 10926 to (510.57, 534.38, 200) mm, rotated rx -180 ry 0 rz 160 deg; joints [10.272, 50.783, -4.113, -141.255, 53.656, 154.567]
  Set speed (19.5 mm/s)
  Call Extruder(543.86861)
  MoveL 10927 to (509.77, 534.61, 200) mm, rotated rx 180 ry 0 rz 160 deg; joints [10.318, 50.646, -3.866, -141.255, 53.762, 154.622]
  Set speed (19.5 mm/s)
  Call Extruder(547.32691)
  MoveL 10928 to (508.62, 534.93, 200) mm, rotated rx 180 ry 0 rz 160 deg; joints [10.381, 50.448, -3.507, -141.258, 53.914, 154.705]
  Set speed (19.5 mm/s)
  Call Extruder(551.99361)
  MoveL 10929 to (507.05, 535.27, 200) mm, rotated rx 180 ry 0 rz 160 deg; joints [10.458, 50.176, -3.016, -141.271, 54.118, 154.824]
  Set speed (19.5 mm/s)
  Call Extruder(556.12848)
  MoveL 10930 to (505.64, 535.52, 200) mm, rotated rx 180 ry 0 rz 160 deg; joints [10.52, 49.932, -2.575, -141.291, 54.298, 154.935]
  Set speed (19.5 mm/s)
  Call Extruder(560.31093)
  MoveL 10931 to (504.21, 535.72, 200) mm, rotated rx 180 ry 0 rz 160 deg; joints [10.576, 49.684, -2.126, -141.318, 54.478, 155.053]
  Set speed (19.5 mm/s)
  Call Extruder(562.11720)
  MoveL 10932 to (503.59, 535.79, 200) mm, rotated rx 180 ry 0 rz 160 deg; joints [10.599, 49.576, -1.931, -141.331, 54.556, 155.105]
  Call Extruder(564.38407)
  MoveL 10933 to (502.81, 535.86, 200) mm, rotated rx 180 ry 0 rz 160 deg; joints [10.625, 49.44, -1.685, -141.351, 54.653, 155.172]
  Set speed (19.5 mm/s)
  Call Extruder(567.75487)
  MoveL 10934 to (501.65, 535.94, 200) mm, rotated rx 180 ry 0 rz 160 deg; joints [10.662, 49.237, -1.319, -141.382, 54.795, 155.274]
  Set speed (19.5 mm/s)
  Call Extruder(572.45242)
  MoveL 10935 to (500.03, 535.97, 200) mm, rotated rx 180 ry 0 rz 160 deg; joints [10.704, 48.952, -0.806, -141.436, 54.992, 155.421]
  Set speed (25.0 mm/s)
  Call Extruder(565.95242)
  MoveL 10936 to (500.03, 535.97, 200) mm, rotated rx 180 ry 0 rz 160 deg; joints [10.704, 48.952, -0.806, -141.436, 54.992, 155.421]
  Call M_RunCode(107)
  Call SetRPM(0.0)
  Call M_RunCode(104)
  Call SetRPM(0.0)
  Call M_RunCode(140)
  Call Extruder(1.00000)
  Call Extruder(-1.00000)
  Set speed (5.0 mm/s)
  MoveL 10937 to (500.03, 535.97, 200) mm, rotated rx 180 ry 0 rz 160 deg; joints [10.704, 48.952, -0.806, -141.436, 54.992, 155.421]
  Set speed (1000.0 mm/s)
  Call ExtrusionStop
  MoveL 10938 to (500.03, 535.97, 200) mm, rotated rx 180 ry 0 rz 160 deg; joints [10.704, 48.952, -0.806, -141.436, 54.992, 155.421]
  MoveL 10939 to (500.03, 535.97, 300) mm, rotated rx 180 ry 0 rz 160 deg; joints [10.704, 38.544, -4.293, -133.463, 44.707, 143.134]
  Call M_RunCode(84)
  Call M_RunCode(82)
  Call SetRPM(0.0)
  Call M_RunCode(104)

--- Python program ExtrusionStart ---
# This script allows adding a trace or a spray deposition
#
# Note: Select Esc key or close the RDK project to clear any trace added using this method
# Note: You can pass an ID as first agurment to specify the trace color
#
# Example:
#    SpindleOn(2)           show the trace in blue
#    SpindleOn(red)         show the trace in red
#    SpindleOff             turn off the trace
#
# Note: You can pass the radius of the trace as a second argument
#    SpindleOn(2,2.5)       show the trace in blue with a sphere of radius 2.5 mm
#
# --------------------------------------------------------------
# This script shows how to create "spray" object in RoboDK that allows simulating particle deposition by using:
# RDK.Spray_Add(tool, object, options_command, volume, geometry)
#    tool: tool item (TCP) to use
#    object: object to project the particles
#    options_command (optional): string to specify options.
#    volume (optional): Matrix of parameters defining the volume of the spray gun
#    geometry (optional): Matrix of vertices defining the triangles.
#
# More information here:
# https://robodk.com/doc/en/PythonAPI/robolink.html#robolink.Robolink.Spray_Add
# https://robodk.com/doc/en/RoboDK-API.html
#
# The scripts ArcStart, ArcEnd and WeldOn and SpindleOn behave in a similar way, the only difference is the default behavior
# This behavior simmulates Fanuc Arc Welding and triggers appropriate output when using the customized post processor.
# Select ESC to clear the trace manually.
#
# Example scripts that use Spray_Add:
#     SpindleOn / SpindleOff    -> Turn trace On/Off
#     ArcOn / ArcOff            -> Turn trace On/Off
#     SprayOn / SprayOff        -> Simulate a spray given a workspace volume (for painting)
#     WeldOn / WeldOff          -> Support for multiple weld guns

#------------------------------------------------------------------
# Set the tool name as shown in the RoboDK tree (set to None to automatically detect)
TOOL_NAME = "ExtruderTool"
# TOOL_NAME = "Spindle"

# Set the part name as shown in the RoboDK tree (set to None to automatically detect)
PART_NAME = "Simple Vase"
# PART_NAME = "Object"

# Radius of the sphere
SPHERE_RADIUS = 3

# Set the particle color as a named color or as AARRGGBB (alpha channel goes first!)
COLOR = "white"
#COLOR = "green"
#COLOR = "#ffff55bb" # pink-red

# Color list to use if we provide an argument
# Example:
#    SpindleOn(2) will show blue
#    SpindleOn(red) will show red
COLOR_LIST = [COLOR, "red", "green", "blue", "cyan", "magenta", "#ffff55bb"]

#------------------------------------------------------------------
import sys # allows getting the passed argument parameters
from robodk import robolink
# Start the RoboDK API
RDK = robolink.Robolink()

# If an arguments from the object events are provided, retrieve the argument
# (index 0 is the file name)
# Use argument index 1 as color index or named color
if len(sys.argv) >= 2:
    # Use argument 1 as color ID if it is numeric
    arg_1 = sys.argv[1]
    if arg_1.isnumeric():
        color_id = int(arg_1)
        if color_id >= 0:
            color_id = color_id % len(COLOR_LIST)
            COLOR = COLOR_LIST[color_id]
    else:
        # Use the named color (or # color)
        COLOR = arg_1

# Use argument index 2 to set the radius
if len(sys.argv) >= 3:
    # Use argument 1 as color ID if it is numeric
    arg_2 = sys.argv[2]
    try:
        SPHERE_RADIUS = float(arg_2)
    except:
        print("Unable to read paramter 2 as radius");

#------------------------------------------------------------------

# Stop if we are not simulating
if RDK.RunMode() != robolink.RUNMODE_SIMULATE:
    quit()

# Create a new spray gun
tool = 0  # auto detect active tool
object = 0 # auto detect object to attach particles

# Use specific tool and part if we provided it
if TOOL_NAME is not None:
    tool = RDK.Item(TOOL_NAME, robolink.ITEM_TYPE_TOOL)

if PART_NAME is not None:
    object = RDK.Item(PART_NAME, robolink.ITEM_TYPE_OBJECT)


# Create a new object with a spray gun
RDK.Spray_Add(tool, object, "PARTICLE=SPHERE(%.2f) NO_PROJECT COLOR=%s" % (SPHERE_RADIUS, COLOR)) # Do not project
# RDK.Spray_Add(tool, object, "PARTICLE=SPHERE(4) PROJECT") # Project to part
RDK.Spray_SetState(robolink.SPRAY_ON)


# Option to use a spread
# coordinates must be provided with respect to the TCP
#close_p0 = [   0,   0, -200] # xyz in mm: Center of the conical ellypse (side 1)
#close_pA = [   5,   0, -200] # xyz in mm: First vertex of the conical ellypse (side 1)
#close_pB = [   0,  10, -200] # xyz in mm: Second vertex of the conical ellypse (side 1)
#close_color = [ 1, 1, 1, 1]  # RGBA (0-1)

#far_p0   = [   0,   0,  50] # xyz in mm: Center of the conical ellypse (side 2)
#far_pA   = [  60,   0,  50] # xyz in mm: First vertex of the conical ellypse (side 2)
#far_pB   = [   0, 120,  50] # xyz in mm: Second vertex of the conical ellypse (side 2)
#far_color   = [ 1, 1, 1, 1]  # RGBA (0-1)

#RDK.Spray_Add(tool, obj, "PARTICLE=CUBE(10,10,2) STEP=8x8")
#RDK.Spray_Add(tool, obj, "PARTICLE=SPHERE(4,8) STEP=8x8")
#RDK.Spray_Add(tool, obj, "PARTICLE=SPHERE(4,8,1,1,0.1) STEP=8x8 RANDX=3")
#RDK.Spray_Add(tool, obj, "PARTICLE=SPHERE(4,8) NO_PROJECT")
#RDK.Spray_Add(tool, obj, "PARTICLE=SPHERE(4,8) STEP=1x0")
#RDK.Spray_Add(tool, obj, "STEP=8x8 RANDX=3", volume.tr(), geom.tr())
#RDK.Spray_SetState(SPRAY_ON)


# Available options:
#     STEP=AxB: Defines the grid to be projected 1x1 means only one line of particle projection (for example, for welding)
#     PARTICLE: Defines the shape and size of particle (sphere or particle), unless a specific geometry is provided:
#       a- SPHERE(radius, facets)
#       b- SPHERE(radius, facets, scalex, scaley, scalez)
#       b- CUBE(sizex, sizey, sizez)
#     RAND=factor: Defines a random factor factor 0 means that the particles are not deposited randomly
#     ELLYPSE: defines the volume as an ellypse (default)
#     RECTANGLE: defines the volume as a rectangle
#     PROJECT: project the particles to the surface (default) (for welding, painting or scanning)
#     NO_PROJECT: does not project the particles to the surface (for example, for 3D printing)

--- Python program ExtrusionStop ---
# This script allows adding a trace or a spray deposition
# More information here:
# https://robodk.com/doc/en/PythonAPI/robolink.html#robolink.Robolink.Spray_Add
#
# Example scripts that use Spray_Add:
#     SpindleOn / SpindleOff    -> Turn trace On/Off
#     ArcOn / ArcOff            -> Turn trace On/Off
#     SprayOn / SprayOff        -> Simulate a spray given a workspace volume (for painting)
#     WeldOn / WeldOff          -> Support for multiple weld guns
#
# Note: Select Esc key or close the RDK project to clear any trace added using this method
# Note: You can pass an ID as first agurment to specify the trace color
#
# Example:
#    SpindleOn(2)           show the trace in blue
#    SpindleOn(red)         show the trace in red
#    SpindleOff             turn off the trace
#
# Note: You can pass the radius of the trace as a second argument
#    SpindleOn(2,2.5)       show the trace in blue with a sphere of radius 2.5 mm
# ---------------------------------------------------------------
#
import sys                # allows getting the passed argument parameters
from robodk import robolink
RDK = robolink.Robolink()

# quit if we are not simulating
if RDK.RunMode() != robolink.RUNMODE_SIMULATE:
    quit()

# Stop the trace
RDK.Spray_SetState(robolink.SPRAY_OFF)
